(* CoDeSys 2.3 export: test2.exp *)
(* Libraries: ANALYZATION.LIB 5.10.99 09:05:06, IECSFC.LIB 13.4.06 15:51:28, STANDARD.LIB 4.10.05 11:14:46 *)

(* PLC configuration (modules and I/O channels)
PLC110_30 [Root] node -1, in %IB0 out %QB0 {param 1 = PLC110-30_v2; param 2 = 1; param 3 = 1000}
  Fast discrete inputs [I_SIMPLE_INPUT] node 0, in %IB0 out %QB0 {param 1 = Fast discrete inputs; param 2 = 10000}
    AT %IX0.0 [BitInput] Discrete input 1 {param 1 = Enter name}
    AT %IX0.1 [BitInput] Discrete input 2 {param 1 = Enter name}
  Discrete inputs - 16 [ID130] node 1, in %IB1 out %QB1 {param 1 = Discrete inputs; param 2 = 10; param 3 = 16}
    AT %IB1.0 [ByteInput] 8 discrete inputs {param 1 = Enter name}
    AT %IB1.1 [ByteInput] 8 discrete inputs {param 1 = Enter name}
  Fast discrete outputs [OWEN_ID570] node 2, in %IB2 out %QB2 {param 1 = Fast discrete outputs; param 2 = FALSE; param 3 = FALSE; param 4 = FALSE; param 5 = FALSE}
    AT %QX2.0 [BitOutput] Fast discrete output 1 {param 1 = Enter name}
    AT %QX2.1 [BitOutput] Fast discrete output 2 {param 1 = Enter name}
    AT %QX2.2 [BitOutput] Fast discrete output 3 {param 1 = Enter name}
    AT %QX2.3 [BitOutput] Fast discrete output 4 {param 1 = Enter name}
  Discrete outputs - 8 [ID131] node 3, in %IB3 out %QB3 {param 1 = Discrete outputs; param 2 = 0; param 3 = No; param 4 = 10}
    AT %QB3.0 [ByteOutput] 8 discrete outputs {param 1 = Enter name}
  Special input [ID103] node 4, in %IB4 out %QB4 {param 1 = Special input}
    AT %IX4.0 [BitInput] Special input {param 1 = Enter name}
  Special output [ID104] node 5, in %IB5 out %QB5 {param 1 = Special output}
    AT %QX5.0 [BitOutput] Special output {param 1 = Enter name}
  ModBus (Master) [MODBUS_MASTER_ID450] node 6, in %IB6 out %QB6 {param 1 = ModBus (Master); param 2 = No}
    AT %QD6.0 [DWordOutput] Last address {param 1 = Enter name}
    AT %QW6.1 [WordOutput] Last error {param 1 = Enter name}
    RS-485-1 [COM1_USART] node 0, in %IB6.0 out %QB6.0 {param 1 = RS-485-1; param 2 = 9600; param 3 = NO PARITY CHECK; param 4 = 8 bits; param 5 = One stop bit; param 6 = RS485; param 7 = RTU; param 8 = 200; param 9 = No}
    Universal Modbus device [ID2000] node 1, in %IB6.1 out %QB6.1 {param 1 = ESP8266; param 2 = 10:0:0:223; param 3 = 150; param 4 = 502; param 5 = Serial; param 6 = 1; param 7 = By poll time; param 8 = 100; param 9 = No; param 10 = 0; param 11 = Trace_mode}
      AT %QB6.1.0 [ComChannel] Command (0xff - Start) {param 1 = Enter name}
      Register output module [ID2004] node 0, in %IB6.1.0 out %QB6.1.0 {param 1 = Register; param 2 = 0; param 3 = Write multiple registers(0x10); param 8 = No}
        mb_out_DefaultTarget AT %QW6.1.0.0 [WordOutput] {param 1 = Enter name}
      Register output module [ID2004] node 1, in %IB6.1.1 out %QB6.1.1 {param 1 = Register; param 2 = 1; param 3 = Write multiple registers(0x10); param 8 = No}
        mb_out_CurrentAngle AT %QW6.1.1.0 [WordOutput] {param 1 = Enter name}
      Register output module [ID2004] node 2, in %IB6.1.2 out %QB6.1.2 {param 1 = Register; param 2 = 2; param 3 = Write multiple registers(0x10); param 8 = No}
        mb_out_TargetAngle AT %QW6.1.2.0 [WordOutput] {param 1 = Enter name}
      Register output module [ID2004] node 3, in %IB6.1.3 out %QB6.1.3 {param 1 = Register; param 2 = 3; param 3 = Write multiple registers(0x10); param 8 = No}
        mb_out_Cycle AT %QW6.1.3.0 [WordOutput] {param 1 = Enter name}
      Register output module [ID2004] node 4, in %IB6.1.4 out %QB6.1.4 {param 1 = Register; param 2 = 4; param 3 = Write multiple registers(0x10); param 8 = No}
        mb_out_Done AT %QW6.1.4.0 [WordOutput] {param 1 = Enter name}
      Register output module [ID2004] node 5, in %IB6.1.5 out %QB6.1.5 {param 1 = Register; param 2 = 5; param 3 = Write multiple registers(0x10); param 8 = No}
        mb_out_Mode AT %QW6.1.5.0 [WordOutput] {param 1 = Enter name}
      Register output module [ID2004] node 6, in %IB6.1.6 out %QB6.1.6 {param 1 = Register; param 2 = 6; param 3 = Write multiple registers(0x10); param 8 = No}
        mb_out_Pedals AT %QW6.1.6.0 [WordOutput] {param 1 = Enter name}
      Register input module [ID2003] node 7, in %IB6.1.7 out %QB6.1.7 {param 1 = Register input module; param 2 = 9; param 3 = Read holding Registers  (0x03); param 8 = No}
        mb_in_Command AT %QW6.1.7.0 [WordOutput] {param 1 = Enter name}
      Register input module [ID2003] node 10, in %IB6.1.10 out %QB6.1.10 {param 1 = Register input module; param 2 = 10; param 3 = Read holding Registers  (0x03); param 8 = No}
        mb_in_WebTarget AT %QW6.1.10.0 [WordOutput] {param 1 = Enter name}
*)

(* Global variable list: Global_Variables *)
VAR_GLOBAL RETAIN
    (* Inputs *)
    gDI_1   AT %IX0.0   : BOOL; (* Fast Input 1 *)
    gDI_2   AT %IX0.1   : BOOL; (* Fast Input 2 *)
    gDI_3   AT %IX1.0.0 : BOOL; (* Input 3 *)
    gDI_4   AT %IX1.0.1 : BOOL; (* Input 4 *)
    gDI_5   AT %IX1.0.2 : BOOL; (* Input 5 *)
    gDI_6   AT %IX1.0.3 : BOOL; (* Input 6 *)
    gDI_7   AT %IX1.0.4 : BOOL; (* Input 7 *)
    gDI_8   AT %IX1.0.5 : BOOL; (* Input 8 *)
    gDI_9   AT %IX1.0.6 : BOOL; (* Input 9 *)
    gDI_10  AT %IX1.0.7 : BOOL; (* Input 10 *)
    gDI_11  AT %IX1.1.0 : BOOL; (* Input 11 *)
    gDI_12  AT %IX1.1.1 : BOOL; (* Input 12 *)
    gDI_13  AT %IX1.1.2 : BOOL; (* Input 13 *)
    gDI_14  AT %IX1.1.3 : BOOL; (* Input 14 *)
    gDI_15  AT %IX1.1.4 : BOOL; (* Input 15 *)
    gDI_16  AT %IX1.1.5 : BOOL; (* Input 16 *)
    gDI_17  AT %IX1.1.6 : BOOL; (* Input 17 *)
    gDI_18  AT %IX1.1.7 : BOOL; (* Input 18 *)

    (* Fast encoder inputs (alias to fast inputs) - keep names used by code *)
    gEncoderA AT %IX0.0 : BOOL;  (* Encoder A (fast input) *)
    gEncoderB AT %IX0.1 : BOOL;  (* Encoder B (fast input) *)

    (* Outputs *)
    gDO_1   AT %QX2.0   : BOOL; (* Fast Output 1 *)
    gDO_2   AT %QX2.1   : BOOL; (* Fast Output 2 *)
    gDO_3   AT %QX2.2   : BOOL; (* Fast Output 3 *)
    gDO_4   AT %QX2.3   : BOOL; (* Fast Output 4 *)

    gDO_5   AT %QX3.0.0 : BOOL; (* Relay/Slow Output 5 *)
    gDO_6   AT %QX3.0.1 : BOOL; (* Relay/Slow Output 6 *)
    gDO_7   AT %QX3.0.2 : BOOL; (* Relay/Slow Output 7 *)
    gDO_8   AT %QX3.0.3 : BOOL; (* Relay/Slow Output 8 *)
    gDO_9   AT %QX3.0.4 : BOOL; (* Relay/Slow Output 9 *)
    gDO_10  AT %QX3.0.5 : BOOL; (* Relay/Slow Output 10 *)
    gDO_11  AT %QX3.0.6 : BOOL; (* Relay/Slow Output 11 *)
    gDO_12  AT %QX3.0.7 : BOOL; (* Relay/Slow Output 12 *)

    (* System outputs *)
    gBeeper AT %QX5.0   : BOOL; (* External beeper output *)

    (* ModBus (Master) system/channel variables exposed by device configuration *)
    gModbus_Master_Channel AT %QD6.0 : DWORD; (* ModBus Master: channel/last address (Q area) *)
    gModbus_Master_LastError AT %QW6.1 : WORD; (* ModBus Master: last error code (Q area) *)

    (* Variables for Modbus and internal state (no AT) *)
    gTargetAngle : REAL := 45.0;    (* target angle, degrees *)
    gDefaultTarget : REAL := 45.0;  (* retained default target; used to toggle between endpoints *)
    gCurrentAngle : REAL := 0.0;    (* current angle, degrees *)
    gCycle : INT := 1;              (* 1=to default, 2=to zero *)
    gAngleFromStart : REAL := 0.0;  (* angle from program start *)
    gStatus : INT := 0;             (* 0=Stop,1=Moving,2=In position *)
    gErrorCode : INT := 0;          (* 0=OK,1=Timeout,2=Fault *)
    gCommand : INT := 0;            (* 1=Start,2=Stop,3=Calibrate *)
    gEncoderCount : DINT := 0;     (* encoder counter for Modbus *)

    (* Calibration / Modbus helper variables *)
    gStartCalib : BOOL := FALSE;
    gCalibRunning : BOOL := FALSE;
    gCalibStatus : INT := 0;
    gCalibRevsDone : INT := 0;
    gCalibRevsTarget : INT := 3;
    gCalibMeasured : REAL := 0.0;
    gCalibCountsPerRev : DINT := 0;
    (* Modbus mapped variables are provided by device configuration channels *)
END_VAR

(* Data type *)
TYPE COMSETTINGS_FALLBACK : STRUCT
    Port : INT; (* PORTS in library; INT used locally to avoid enum conflicts *)
    dwBaudRate : DWORD;
    byStopBits : BYTE;
    byParity : BYTE;
    dwTimeout : DWORD;
    dwBufferSize : DWORD;
    dwScan : DWORD;
END_STRUCT
END_TYPE

(* POU PLC_PRG, ST *)
PROGRAM PLC_PRG
VAR
    (* Логика режима и кнопок *)
    prev_d5 : BOOL := TRUE;
    enableStart : BOOL;      (* D5: 1-ручной, 0-авто *)
    btnD7 : BOOL;            (* D7: педаль вперед *)
    btnD8 : BOOL;            (* D8: педаль назад *)
    both : BOOL;             (* Обе нажаты *)
    
    (* Детекторы фронтов *)
    encAEdge : R_TRIG;
    encBEdge : R_TRIG;
    
    (* Состояние цикла *)
    done : BOOL := FALSE;    (* Флаг завершения гиба *)
    
    (* Таймеры и сигналы *)
    targetPulseTrigger : BOOL := FALSE;
    tpTarget : TP;           (* Импульс на DO12 *)
    beepTargetTrigger : BOOL := FALSE;
    tpBeepTarget : TP;       (* Писк при достижении цели *)
    
    errorBeepTrigger : BOOL := FALSE;
    tErrTotal : TON;
    tErrDelay1 : TON;
    tErrDelay2 : TON;
    tErrDelay3 : TON;
    rTrigErr1 : R_TRIG;
    rTrigErr2 : R_TRIG;
    rTrigErr3 : R_TRIG;
    tpErr : TP;

    (* Память для логики фронтов *)
    prev_d7 : BOOL := FALSE;
    prev_d8 : BOOL := FALSE;
    prev_both : BOOL := FALSE;

    (* Modbus переменные *)
    prev_mb_in_command : WORD := 0;
END_VAR
(* 1. ЧТЕНИЕ ФИЗИЧЕСКИХ ВХОДОВ *)
enableStart := gDI_5; 
btnD7 := gDI_7;       
btnD8 := gDI_8;       
both := btnD7 AND btnD8;

(* 2. ОБРАБОТКА ЭНКОДЕРА *)
encAEdge(CLK := gEncoderA);
encBEdge(CLK := gEncoderB);

IF encAEdge.Q THEN
    IF gEncoderB THEN
        gEncoderCount := gEncoderCount + 1;
    ELSE
        gEncoderCount := gEncoderCount - 1;
    END_IF;
END_IF;

(* 3. РАСЧЕТ ТЕКУЩЕГО УГЛА *)
IF (gCalibCountsPerRev = 0) THEN
    gCalibCountsPerRev := 360;
END_IF;
gCurrentAngle := - DINT_TO_REAL(gEncoderCount) * 360.0 / DINT_TO_REAL(gCalibCountsPerRev);

(* 4. КАЛИБРОВКА НОЛЯ ПРИ ПЕРЕХОДЕ В АВТО *)
IF (prev_d5 AND NOT enableStart) THEN
    gEncoderCount := 0;
    gCurrentAngle := 0.0;
    gCycle := 1;
    gTargetAngle := gDefaultTarget;
    done := FALSE;
END_IF;
prev_d5 := enableStart;

(* 5. ПРИЕМ ДАННЫХ ИЗ ВЕБА (ESP -> PLC) *)

(* Чтение целевого угла (Регистр 10) *)
IF mb_in_WebTarget <> 0 THEN
    IF ABS(gTargetAngle - (WORD_TO_REAL(mb_in_WebTarget) / 10.0)) > 0.1 THEN
        gTargetAngle := WORD_TO_REAL(mb_in_WebTarget) / 10.0;
        gDefaultTarget := gTargetAngle; 
        done := FALSE; 
    END_IF;
END_IF;

(* Чтение команд Старт/Стоп/Ноль (Регистр 9) *)
IF mb_in_Command <> 0 AND mb_in_Command <> prev_mb_in_command THEN
    CASE WORD_TO_INT(mb_in_Command) OF
        1: (* СТАРТ *)
            IF NOT enableStart THEN done := FALSE; gCycle := 1; END_IF;
        2: (* СТОП *)
            done := TRUE; (* Режим "Стоп" - имитируем достижение цели *)
        3: (* НОЛЬ *)
            gEncoderCount := 0; gCurrentAngle := 0.0;
    END_CASE;
END_IF;
prev_mb_in_command := mb_in_Command;

(* 6. ВЫБОР ЦЕЛИ В ЗАВИСИМОСТИ ОТ ЦИКЛА (АВТО) *)
IF NOT enableStart AND NOT done THEN
    IF gCycle = 1 THEN
        gTargetAngle := gDefaultTarget;
    ELSIF gCycle = 2 THEN
        gTargetAngle := 0.0;
    END_IF;
END_IF;

(* 7. ОТПРАВКА ДАННЫХ В ВЕБ (PLC -> ESP) *)
mb_out_DefaultTarget := REAL_TO_WORD(gDefaultTarget * 10.0);
mb_out_CurrentAngle  := REAL_TO_WORD(ABS(gCurrentAngle * 10.0));
mb_out_TargetAngle   := REAL_TO_WORD(gTargetAngle * 10.0);
mb_out_Cycle         := INT_TO_WORD(gCycle);

IF done THEN mb_out_Done := 1; ELSE mb_out_Done := 0; END_IF;
IF enableStart THEN mb_out_Mode := 1; ELSE mb_out_Mode := 0; END_IF;

mb_out_Pedals := 0;
IF btnD7 THEN mb_out_Pedals := mb_out_Pedals + 1; END_IF;
IF btnD8 THEN mb_out_Pedals := mb_out_Pedals + 2; END_IF;

(* 8. ЛОГИКА УПРАВЛЕНИЯ МОТОРОМ *)
IF enableStart THEN  (* Ручной режим *)
    gDO_10 := btnD7 AND NOT btnD8 AND NOT both;
    gDO_11 := btnD8 AND NOT btnD7 AND NOT both;
ELSE  (* Авто режим *)
    gDO_10 := btnD7 AND NOT btnD8 AND (gCurrentAngle < gTargetAngle) AND NOT done;
    gDO_11 := btnD8 AND NOT btnD7 AND (gCurrentAngle > 0.0) AND NOT done;
END_IF;

(* 9. АВТОМАТИЧЕСКИЙ ОСТАНОВ *)
IF NOT enableStart AND NOT done THEN
    IF (ABS(gCurrentAngle - gTargetAngle) < 0.5) THEN
        done := TRUE;
        targetPulseTrigger := TRUE;
        beepTargetTrigger := TRUE;
        IF gCycle = 1 THEN gCycle := 2; ELSE gCycle := 1; END_IF;
    END_IF;
END_IF;

(* Если вручную или через веб угол ушел от цели - сбрасываем Done *)
IF (ABS(gCurrentAngle - gTargetAngle) > 2.0) THEN
    done := FALSE;
END_IF;

(* 10. ОБРАБОТКА ТАЙМЕРОВ И СИГНАЛОВ (ИСПРАВЛЕНО) *)
tpTarget(IN := targetPulseTrigger, PT := T#500MS);
gDO_12 := tpTarget.Q;
IF tpTarget.Q THEN targetPulseTrigger := FALSE; END_IF;

tpBeepTarget(IN := beepTargetTrigger, PT := T#500MS);
(* Сигнал ошибки *)
IF NOT enableStart AND NOT done THEN
    IF ((btnD7 AND NOT prev_d7) AND (gCurrentAngle >= gDefaultTarget)) OR
       ((btnD8 AND NOT prev_d8) AND (gCurrentAngle <= 0.0)) OR
       (both AND NOT prev_both) THEN
        errorBeepTrigger := TRUE;
    END_IF;
END_IF;

tErrTotal(IN := errorBeepTrigger, PT := T#1400MS);
tErrDelay1(IN := errorBeepTrigger, PT := T#0MS);
tErrDelay2(IN := errorBeepTrigger, PT := T#400MS);
tErrDelay3(IN := errorBeepTrigger, PT := T#800MS);
rTrigErr1(CLK := tErrDelay1.Q);
rTrigErr2(CLK := tErrDelay2.Q);
rTrigErr3(CLK := tErrDelay3.Q);
tpErr(IN := (rTrigErr1.Q OR rTrigErr2.Q OR rTrigErr3.Q), PT := T#200MS);

gBeeper := tpBeepTarget.Q OR tpErr.Q;

IF tErrTotal.Q THEN errorBeepTrigger := FALSE; END_IF;

prev_d7 := btnD7;
prev_d8 := btnD8;
prev_both := both;
END_PROGRAM
